FUNCTION FC_Current4_20Raw_TO_Percentage : REAL
VAR_INPUT
	i : REAL;
END_VAR
VAR
	f : REAL;
	nIntMax : REAL := 32767;
	nIntMin : REAL := 6553;
END_VAR

FC_Current4_20Raw_TO_Percentage := 100*(i-nIntMin)/(nIntMax-nIntMin);

END_FUNCTION

(* stored: Version 1.1.0.1, ProductVersion 3.1.4024.3
   POU FC_Current4_20Raw_TO_Percentage: Id {dd630bbf-9024-486e-8a7e-a3259ba9082e}, SpecialFunc None *)
